INTERFACE ITF_Valve

END_INTERFACE

(* stored: Version 1.1.0.1
   Itf ITF_Valve: Id {0d54bfdc-bb88-4a13-810b-36b059e132df} *)
